{attribute 'qualified_only'}
VAR_GLOBAL
    TestRunner : TTestRunner;
    
END_VAR

(* stored: Version 1.1.0.1, ProductVersion 3.1.4024.3
   GVL TestFramework: Id {ca7c940a-60ec-4292-9382-a233f6d36546} *)
